// TwinCAT 3 PLC project Fundamentals
// ProgramVersion: 3.1.4023.0
// libraries:
//   Tc2_Standard, * (Beckhoff Automation GmbH)
//   Tc2_System, * (Beckhoff Automation GmbH)
//   Tc2_Utilities, * (Beckhoff Automation GmbH)
//   Tc3_Module, * (Beckhoff Automation GmbH)
// project tree:
//   DUTs/ Breakout.TcDUT
//   DUTs/Simulator/ Compass.TcDUT, Intersection.TcDUT, TrafficDensity.TcDUT, TrafficLight.TcDUT
//   GVLs/ Comparison_GVL.TcGVL, Traffic_GVL.TcGVL
//   / PlcTask.TcTTO
//   POUs/HandsOnProject/ Cars.TcPOU, TrafficManager.TcPOU, TrafficLights.TcPOU
//   POUs/Kim%27s Solution/ Kims_UpdateLights.TcPOU (not stored)
//   POUs/ Ladder.TcPOU, MAIN.TcPOU, StructuredText.TcPOU
// real-time tasks:
//   TASK PlcTask: cycle T#2ms, priority 20, ADS port 350
//   TASK PlcTask1: cycle T#2ms, priority 21, ADS port 351
// I/O:
//   DEVICE Device 1 (EtherCAT), AmsNetId 172.30.193.100.2.1
//     Term 1 (EK1200) [EK1200-5000 EtherCAT Power supply (2A E-Bus)]
//       Term 2 (EL6900) [EL6900, TwinSAFE PLC]
//       Term 3 (EL1904) [EL1904, 4 Ch. Safety Input 24V, TwinSAFE]
//         modules: Module 1 (FSOES)
//       Term 4 (EL2904) [EL2904, 4 Ch. Safety Output 24V, 0.5A, TwinSAFE]
//         modules: Module 1 (FSOES), Module 2 (DO)
//       Term 5 (EL1008) [EL1008 8Ch. Dig. Input 24V, 3ms]
//       Term 6 (EL2008) [EL2008 8Ch. Dig. Output 24V, 0.5A]
//       Term 7 (EL1008) [EL1008 8Ch. Dig. Input 24V, 3ms]
//       Term 8 (EL2008) [EL2008 8Ch. Dig. Output 24V, 0.5A]
//       Term 9 (EL9410) [EL9410 E-Bus Power Supplier  (Diagnostics)]
//       Term 10 (EL1008) [EL1008 8Ch. Dig. Input 24V, 3ms]
//       Term 11 (EL2008) [EL2008 8Ch. Dig. Output 24V, 0.5A]
//       Term 12 (EL1008) [EL1008 8Ch. Dig. Input 24V, 3ms]
//       Term 13 (EL2008) [EL2008 8Ch. Dig. Output 24V, 0.5A]
//       Term 14 (EL1008) [EL1008 8Ch. Dig. Input 24V, 3ms]
//       Term 15 (EL2008) [EL2008 8Ch. Dig. Output 24V, 0.5A]
//       Term 16 (EL9011) [EL9011 End Terminal]
//   DEVICE Device 4 (EtherCAT), AmsNetId 172.30.193.100.5.1
//     Drive 17 (Elmo Drive ) [Gold EtherCAT GCON Drive Rev:0x00010420]
//     Drive 18 (Elmo Drive ) [Gold EtherCAT GCON Drive Rev:0x00010420]
//     Drive 19 (Elmo Drive ) [Gold EtherCAT GCON Drive Rev:0x00010420]
//     Drive 20 (Elmo Drive ) [Gold EtherCAT GCON Drive Rev:0x00010420]
//     Drive 21 (Elmo Drive ) [Gold EtherCAT GCON Drive Rev:0x00010420]
//     Drive 22 (Elmo Drive ) [Gold EtherCAT GCON Drive Rev:0x00010420]

CONFIGURATION Fundamentals
    RESOURCE PLC ON TwinCAT3
        TASK PlcTask(INTERVAL := T#2ms, PRIORITY := 20);
        PROGRAM MAIN WITH PlcTask : MAIN;
    END_RESOURCE
END_CONFIGURATION

// ---- DUTs/Breakout.TcDUT
	{attribute 'OPC.UA.DA' := '1'}
	{attribute 'OPC.UA.DA.StructuredType' := '1'}
TYPE Breakout :
STRUCT
	RedLight	AT %Q*:BOOL; 
	AmberLight	AT %Q*:BOOL;
	GreenLight	AT %Q*:BOOL;
	BlueLight  	AT %Q*:BOOL;
	ButtonPushed AT %I*:BOOL;
END_STRUCT
END_TYPE

// ---- DUTs/Simulator/Compass.TcDUT
{attribute 'strict'}
TYPE Compass :
(
	North:= 1,
	South:= 2,
	East:= 3,
	West:= 4
);
END_TYPE

// ---- DUTs/Simulator/Intersection.TcDUT
	{attribute 'OPC.UA.DA' := '1'}
	{attribute 'OPC.UA.DA.StructuredType' := '1'}
TYPE Intersection :
STRUCT
	NS_Road: TrafficDensity ;//  Values: None/Low/Medium/High
	EW_Road: TrafficDensity ;// Values: None/Low/Medium/High
	
	//The traffic lights facing each direction (N_Light.Red := True -> turns the red light on for traffic flowing North to South);
	N_Light: TrafficLight; //.Red .Amber .Green
	S_Light: TrafficLight; //.Red .Amber .Green
	W_Light: TrafficLight; //.Red .Amber .Green
	E_Light: TrafficLight; //.Red .Amber .Green
	
	//pedestrian crossing request buttons
	N_Ped AT %I*: BOOL;
	S_Ped AT %I*: BOOL;
	E_Ped AT %I*: BOOL;
	W_Ped AT %I*: BOOL;
	
	//Pedestrian safe to cross indicator (the blue light)
	N_Cross AT %Q*: BOOL;
	S_Cross AT %Q*: BOOL;
	E_Cross AT %Q*: BOOL;
	W_Cross AT %Q*: BOOL;
	//Does this direction lead out of the area
	Exit1, Exit2: Compass; //1-4 N S E W
	
	//Stores presense of cars in each direction of the intersection, filled and emptied by the simulation logic
	CarQueue: ARRAY[1..4] OF INT; //1-4 N S E W
END_STRUCT
END_TYPE

// ---- DUTs/Simulator/TrafficDensity.TcDUT
{attribute 'qualified_only'}
{attribute 'OPC.UA.DA' := '1'}
{attribute 'OPC.UA.DA.StructuredType' := '1'}
TYPE TrafficDensity :
(
	None 	:= 0,
	High	:= 1, //Broadway
	Medium	:= 5, //Brick Church
	Low		:= 10 //Fernco
);
END_TYPE

// ---- DUTs/Simulator/TrafficLight.TcDUT
TYPE TrafficLight :
STRUCT
	Red		AT %Q*:BOOL; 
	Amber	AT %Q*:BOOL;
	Green	AT %Q*:BOOL;
END_STRUCT
END_TYPE

// ---- GVLs/Comparison_GVL.TcGVL
{attribute 'qualified_only'} 
VAR_GLOBAL
	NormallyOpen_NO	: BOOL;
	NormallyClosed_NC : BOOL;
	This_And		: BOOL;
	This_Or			: BOOL;
	Or_This			: BOOL;
	Or_NOT_This		: BOOL:=TRUE;
	But_NOT_This	: BOOL:=TRUE;
	And_This		: BOOL;
	Tada			: BOOL;
	OffTimer_TOF	: TOF;
	OnTimer_TON		: TON;
	PulseTimer_TP	: TP;
	TurnOFFAfter	: BOOL;
	TurnONAfter		: BOOL;
	TurnOnFor		: BOOL;
	DefaultON		: BOOL;
	DefaultOFF		: BOOL;
	Countdown		: CTD;
	
	CountUP			: CTU;
	CountTo25		: BOOL;
END_VAR
VAR_GLOBAL CONSTANT
	DURATION		:TIME:=T#15S;
	SHORT_DURATION	:TIME:=T#5S;
END_VAR

// ---- GVLs/Traffic_GVL.TcGVL
VAR_GLOBAL
	{attribute 'OPC.UA.DA' := '1'}
	{attribute 'OPC.UA.DA.StructuredType' := '1'}
	FirstAndMain 	:Intersection;
	{attribute 'OPC.UA.DA' := '1'}
	{attribute 'OPC.UA.DA.StructuredType' := '1'}
	SecondAndMain 	:Intersection;
	{attribute 'OPC.UA.DA' := '1'}
	{attribute 'OPC.UA.DA.StructuredType' := '1'}
	FirstAndPine	:Intersection;
	{attribute 'OPC.UA.DA' := '1'}
	{attribute 'OPC.UA.DA.StructuredType' := '1'}
	SecondAndPine	:Intersection;
	
END_VAR

// ---- POUs/MAIN.TcPOU
PROGRAM MAIN
VAR
	ClimbTheRungs, MoveOnToCode, PlayInTraffic, RunOnce:BOOL:=FALSE;
	
	{attribute 'OPC.UA.DA' := '1'}
	{attribute 'OPC.UA.DA.StructuredType' := '1'}
	FirstSteps:Breakout;
END_VAR

// <- this is how you comment out lines, anything after the // will not be part of the program 
//this is how you can leave notes for future developers or if code isn't working right you can remove it temporarily to test things without deleting it  

//THIS SPACE IS WHERE YOU CAN PUT YOUR FIRST CODE, Try removing the // from the next line
//FirstSteps.BlueLight := TRUE;


IF ClimbTheRungs THEN
	Ladder(); //This calls the ladder logic example
ELSIF MoveOnToCode THEN
StructuredText(); //This calls the structured text example
ELSIF PlayInTraffic THEN
	IF NOT RunOnce THEN
	TrafficManager.Init();
	runOnce:=TRUE;
END_IF
TrafficManager.Update();
END_IF

END_PROGRAM

// ---- POUs/Ladder.TcPOU
PROGRAM Ladder
VAR

END_VAR
VAR // added by the converter: edge detectors and wires of the graphical bodies
    _rt1 : R_TRIG;
END_VAR

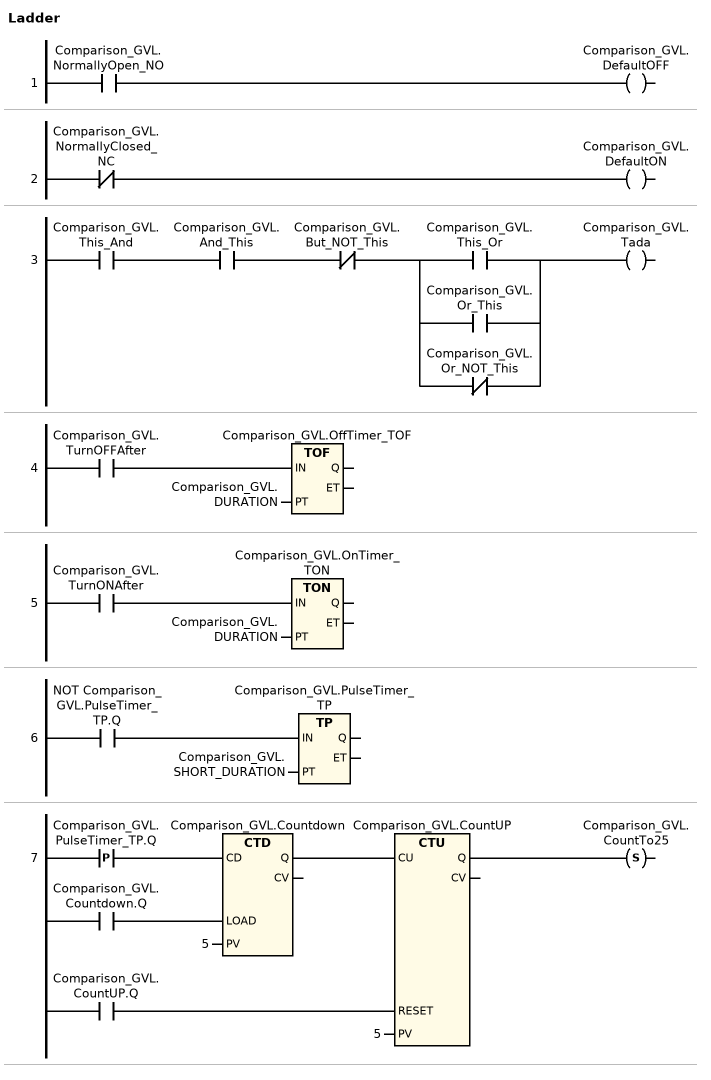
// NETWORK 1
Comparison_GVL.DefaultOFF := Comparison_GVL.NormallyOpen_NO;

// NETWORK 2
Comparison_GVL.DefaultON := NOT Comparison_GVL.NormallyClosed_NC;

// NETWORK 3
Comparison_GVL.Tada := Comparison_GVL.This_And AND Comparison_GVL.And_This AND NOT Comparison_GVL.But_NOT_This AND (Comparison_GVL.This_Or OR Comparison_GVL.Or_This OR NOT Comparison_GVL.Or_NOT_This);

// NETWORK 4
Comparison_GVL.OffTimer_TOF(IN := Comparison_GVL.TurnOFFAfter, PT := Comparison_GVL.DURATION); // TOF

// NETWORK 5
Comparison_GVL.OnTimer_TON(IN := Comparison_GVL.TurnONAfter, PT := Comparison_GVL.DURATION); // TON

// NETWORK 6
Comparison_GVL.PulseTimer_TP(IN := NOT Comparison_GVL.PulseTimer_TP.Q, PT := Comparison_GVL.SHORT_DURATION); // TP

// NETWORK 7
_rt1(CLK := Comparison_GVL.PulseTimer_TP.Q);
Comparison_GVL.Countdown(CD := _rt1.Q, LOAD := Comparison_GVL.Countdown.Q, PV := 5); // CTD
Comparison_GVL.CountUP(CU := Comparison_GVL.Countdown.Q, RESET := Comparison_GVL.CountUP.Q, PV := 5); // CTU
Comparison_GVL.CountTo25 S= Comparison_GVL.CountUP.Q;

END_PROGRAM

// ---- POUs/StructuredText.TcPOU
PROGRAM StructuredText
VAR
	ChangeTime		:TIME:=T#1S;
	CountOnes		:INT:=1;
	CountFives		:INT:=1;
	JustOncePer 	:R_TRIG;
	DidSomething:BOOL;
	AlsoCountTo25	: BOOL;
END_VAR
VAR CONSTANT
	ST_DURATION	:TIME:=T#2S;
END_VAR

	Comparison_GVL.DefaultOFF	:=	Comparison_GVL.NormallyOpen_NO; //Sets DefaultOFF equal to whatever NormallyOpen is set to
	Comparison_GVL.DefaultON	:=	NOT Comparison_GVL.NormallyClosed_NC; //Sets DefaultON equal to the opposite of what NormallyClosed is set to
	
	Comparison_GVL.Tada			:= Comparison_GVL.This_And AND Comparison_GVL.And_This	AND NOT Comparison_GVL.But_NOT_This	AND
								(Comparison_GVL.This_Or OR Comparison_GVL.Or_This OR NOT Comparison_GVL.Or_NOT_This);
	
	// this line ^ and this next one technically do the same thing BUT if I wanted to do more complicated stuff or multiple things I need to use the IF 
	
	IF Comparison_GVL.This_And AND Comparison_GVL.And_This	AND NOT Comparison_GVL.But_NOT_This	AND
		(Comparison_GVL.This_Or OR Comparison_GVL.Or_This OR NOT Comparison_GVL.Or_NOT_This) THEN
		Comparison_GVL.Tada	:= TRUE;
	ELSE
		Comparison_GVL.Tada	:= FALSE;
	END_IF
	
	Comparison_GVL.OffTimer_TOF(IN:=Comparison_GVL.TurnOFFAfter,PT:= ST_DURATION);
	Comparison_GVL.OnTimer_TON(IN:=Comparison_GVL.TurnONAfter,PT:= ST_DURATION);
	Comparison_GVL.PulseTimer_TP(IN:=NOT Comparison_GVL.PulseTimer_TP.Q,PT:= ChangeTime);
	JustOncePer(CLK:= Comparison_GVL.PulseTimer_TP.Q);
	
	IF JustOncePer.Q THEN
		CountOnes:= CountOnes+1;
		Comparison_GVL.TurnOnFor:=FALSE;
	END_IF
	IF CountOnes = 5 THEN
		CountFives:= CountFives +1;
		CountOnes:=1;
	END_IF	
	
	DidSomething:= DoSomething(Counter:= (CountOnes*CountFives) );
	
	IF CountFives = 5 THEN
		CountFives:=1;
	END_IF

METHOD DoSomething : BOOL
VAR_INPUT
	Counter:INT;
END_VAR
CASE Counter OF
	1,10,20:
		Comparison_GVL.TurnOFFAfter:=TRUE;
		Comparison_GVL.TurnONAfter:=TRUE;
		DoSomething:=TRUE;
	2,11,21:
		Comparison_GVL.TurnOFFAfter:=FALSE;
		DoSomething:=TRUE;
	3:
		Comparison_GVL.This_And:=TRUE;
		Comparison_GVL.And_This:=TRUE;
		DoSomething:=TRUE;
	5:
		Comparison_GVL.But_NOT_This:=FALSE;
		DoSomething:=TRUE;
	7:
		Comparison_GVL.This_Or:=TRUE;
		DoSomething:=TRUE;
	9,19:
		Comparison_GVL.TurnONAfter:=FALSE;
		DoSomething:=TRUE;
	13:
		Comparison_GVL.Or_This:=TRUE;
		DoSomething:=TRUE;
	15:
		Comparison_GVL.Or_This:=FALSE;
		Comparison_GVL.Or_NOT_This:=FALSE;
		DoSomething:=TRUE;
	17:
		Comparison_GVL.This_Or:=FALSE;
		Comparison_GVL.Or_This:=FALSE;
		DoSomething:=TRUE;
	25:
		AlsoCountTo25:=TRUE;
	ELSE
		DoSomething:=FALSE;
		Comparison_GVL.TurnOnFor:=TRUE;
END_CASE
END_METHOD

END_PROGRAM

// ---- POUs/HandsOnProject/TrafficManager.TcPOU
PROGRAM TrafficManager
VAR
Simulator: Cars;
UpdateLights: Kims_UpdateLights;
runOnce:BOOL:=FALSE;
END_VAR

METHOD Change_TrafficFlow : BOOL
VAR_INPUT
	Intersect: POINTER to Intersection;
	NewNS_Density, NewEW_Density: TrafficDensity;
	Exit1, Exit2: Compass;
END_VAR
Intersect^.NS_Road:= NewNS_Density;
Intersect^.EW_Road:= NewEW_Density;
Intersect^.Exit1 := Exit1;
Intersect^.Exit2 := Exit2;
END_METHOD

METHOD Init : BOOL
VAR_INPUT
	//First, Second, Main, Pine :TrafficDensity;
END_VAR
//FirstAndMain.NS_Road:=TrafficDensity.Low;
//FirstAndMain.EW_Road:=TrafficDensity.Medium;
//FirstAndMain.Exit1:= North;
//FirstAndMain.Exit2:= West;
Change_TrafficFlow(ADR(FirstAndMain),TrafficDensity.Low,TrafficDensity.Medium, North, West);
Change_TrafficFlow(ADR(SecondAndMain),TrafficDensity.Medium,TrafficDensity.Medium, North, East);

Change_TrafficFlow(ADR(FirstAndPine),TrafficDensity.Low,TrafficDensity.High, South, West);
Change_TrafficFlow(ADR(SecondAndPine),TrafficDensity.Medium,TrafficDensity.High, South, East);
END_METHOD

METHOD Update
VAR_INPUT
END_VAR
UpdateLights(Intersect:=ADR(FirstAndMain));
UpdateLights(Intersect:=ADR(SecondAndMain));
//			  |						   |
//---------------<-Main Street->------------------
//		First |					Second |
//			  |						   |
//			  |  					   |
//----------------<-Pine Street->------------------
//			  |						   |
UpdateLights(Intersect:=ADR(FirstAndPine));
UpdateLights(Intersect:=ADR(SecondAndPine));


//Below this point I'm just Playing with my Hot Wheels haha//
Simulator.AddCars(ADR(FirstAndMain));
Simulator.AddCars(ADR(SecondAndMain));
Simulator.AddCars(ADR(FirstAndPine));
Simulator.AddCars(ADR(SecondAndPine));
Simulator.MoveCars(ADR(FirstAndMain), ADR(SecondAndMain), Compass.East, ADR(FirstAndPine), Compass.South);
Simulator.MoveCars(ADR(SecondAndPine), ADR(SecondAndMain), Compass.North, ADR(FirstAndPine), Compass.West);
END_METHOD

END_PROGRAM

// ---- POUs/HandsOnProject/Cars.TcPOU
FUNCTION_BLOCK Cars
VAR_INPUT
END_VAR
VAR_OUTPUT
END_VAR
VAR
	CarSpawner		:TON;
	SpawnRate		:INT;
END_VAR

METHOD AddCars : BOOL
VAR_INPUT
	Intersect:POINTER TO Intersection;
END_VAR
VAR
	Frequency: TIME := T#1S;
END_VAR
CarSpawner(IN := NOT CarSpawner.Q, PT := Frequency);
IF CarSpawner.Q THEN
	SpawnRate:=SpawnRate+1;
	CASE Intersect^.Exit1 OF
		North, South:
			IF SpawnRate MOD Intersect^.NS_Road = 0 THEN
				Intersect^.CarQueue[Intersect^.Exit1]:= Intersect^.CarQueue[Intersect^.Exit1] +1;
			END_IF		
		East, West:
			IF SpawnRate MOD Intersect^.EW_Road = 0 THEN
				Intersect^.CarQueue[Intersect^.Exit1]:= Intersect^.CarQueue[Intersect^.Exit1] +1;
			END_IF
	END_CASE
	IF NOT (Intersect^.Exit2 = Intersect^.Exit1) THEN
		CASE Intersect^.Exit2 OF	
		North, South:
			IF SpawnRate MOD Intersect^.NS_Road = 0 THEN
				Intersect^.CarQueue[Intersect^.Exit2]:= Intersect^.CarQueue[Intersect^.Exit2] +1;
			END_IF		
		East, West:
			IF SpawnRate MOD Intersect^.EW_Road = 0 THEN
				Intersect^.CarQueue[Intersect^.Exit2]:= Intersect^.CarQueue[Intersect^.Exit2] +1;
			END_IF
		END_CASE	
	END_IF

END_IF
IF SpawnRate = 10 THEN
	SpawnRate :=0;
END_IF
END_METHOD

METHOD MoveCars : BOOL
VAR_INPUT
	To_Intersect, From_A: POINTER TO Intersection;
	Direction_A: Compass;
	From_B: POINTER TO Intersection;
 	Direction_B: Compass;	
END_VAR
//The traffic lights are facing each direction (N_Light.Red := True -> turns the red light facing north on stopping traffic flowing North to South);
IF CarSpawner.Q THEN
	CASE Direction_A OF
	North:
		IF From_A^.N_Light.Green = TRUE AND From_A^.CarQueue[North]>0 THEN
			From_A^.CarQueue[North]:= From_A^.CarQueue[North] - 1;
			IF To_Intersect^.N_Light.Green AND (To_Intersect^.Exit1 = North OR To_Intersect^.Exit2 = North) THEN
				To_Intersect^.CarQueue[North]:= To_Intersect^.CarQueue[North] - 1;
			ELSE
				To_Intersect^.CarQueue[North]:= To_Intersect^.CarQueue[North] + 1;
			END_IF
			
		END_IF
		IF To_Intersect^.S_Light.Green = TRUE AND To_Intersect^.CarQueue[South]>0 THEN
			To_Intersect^.CarQueue[South]:= To_Intersect^.CarQueue[South] - 1;
			IF From_A^.S_Light.Green AND (From_A^.Exit1 = South OR From_A^.Exit2 = South) THEN
				From_A^.CarQueue[South]:= From_A^.CarQueue[South] - 1;
			ELSE
				From_A^.CarQueue[South]:= From_A^.CarQueue[South] + 1;
			END_IF
		END_IF
	South:
		IF From_A^.S_Light.Green = TRUE AND From_A^.CarQueue[South]>0 THEN
			From_A^.CarQueue[South]:= From_A^.CarQueue[South] - 1;
			IF To_Intersect^.S_Light.Green AND (To_Intersect^.Exit1 = South OR To_Intersect^.Exit2 = South) THEN
				To_Intersect^.CarQueue[South]:= To_Intersect^.CarQueue[South] - 1;
			ELSE
				To_Intersect^.CarQueue[South]:= To_Intersect^.CarQueue[SOuth] + 1;
			END_IF
			
		END_IF
		IF To_Intersect^.N_Light.Green = TRUE AND To_Intersect^.CarQueue[North]>0 THEN
			To_Intersect^.CarQueue[North]:= To_Intersect^.CarQueue[North] - 1;
			IF From_A^.N_Light.Green AND (From_A^.Exit1 = North OR From_A^.Exit2 = North) THEN
				From_A^.CarQueue[North]:= From_A^.CarQueue[North] - 1;
			ELSE
				From_A^.CarQueue[North]:= From_A^.CarQueue[North] + 1;
			END_IF
		END_IF
	East:
		IF From_A^.E_Light.Green = TRUE AND From_A^.CarQueue[East]>0 THEN
			From_A^.CarQueue[East]:= From_A^.CarQueue[East] - 1;
			IF To_Intersect^.E_Light.Green AND (To_Intersect^.Exit1 = East OR To_Intersect^.Exit2 = East) THEN
				To_Intersect^.CarQueue[East]:= To_Intersect^.CarQueue[East] - 1;
			ELSE
				To_Intersect^.CarQueue[East]:= To_Intersect^.CarQueue[East] + 1;
			END_IF
			
		END_IF
		IF To_Intersect^.W_Light.Green = TRUE AND To_Intersect^.CarQueue[West]>0 THEN
			To_Intersect^.CarQueue[West]:= To_Intersect^.CarQueue[West] - 1;
			IF From_A^.W_Light.Green AND (From_A^.Exit1 = West OR From_A^.Exit2 = West) THEN
				From_A^.CarQueue[West]:= From_A^.CarQueue[West] - 1;
			ELSE
				From_A^.CarQueue[West]:= From_A^.CarQueue[West] + 1;
			END_IF
		END_IF
	West:
		IF From_A^.W_Light.Green = TRUE AND From_A^.CarQueue[West]>0 THEN
			From_A^.CarQueue[West]:= From_A^.CarQueue[West] - 1;
			IF To_Intersect^.W_Light.Green AND (To_Intersect^.Exit1 = West OR To_Intersect^.Exit2 = West) THEN
				To_Intersect^.CarQueue[West]:= To_Intersect^.CarQueue[West] - 1;
			ELSE
				To_Intersect^.CarQueue[West]:= To_Intersect^.CarQueue[West] + 1;
			END_IF
			
		END_IF
		IF To_Intersect^.E_Light.Green = TRUE AND To_Intersect^.CarQueue[East]>0 THEN
			To_Intersect^.CarQueue[East]:= To_Intersect^.CarQueue[East] - 1;
			IF From_A^.E_Light.Green AND (From_A^.Exit1 = East OR From_A^.Exit2 = East) THEN
				From_A^.CarQueue[East]:= From_A^.CarQueue[East] - 1;
			ELSE
				From_A^.CarQueue[East]:= From_A^.CarQueue[East] + 1;
			END_IF
		END_IF
	END_CASE
		CASE Direction_B OF
	North:
		IF From_B^.N_Light.Green = TRUE AND From_B^.CarQueue[North]>0 THEN
			From_B^.CarQueue[North]:= From_B^.CarQueue[North] - 1;
			IF To_Intersect^.N_Light.Green AND (To_Intersect^.Exit1 = North OR To_Intersect^.Exit2 = North) THEN
				To_Intersect^.CarQueue[North]:= To_Intersect^.CarQueue[North] - 1;
			ELSE
				To_Intersect^.CarQueue[North]:= To_Intersect^.CarQueue[North] + 1;
			END_IF
			
		END_IF
		IF To_Intersect^.S_Light.Green = TRUE AND To_Intersect^.CarQueue[South]>0 THEN
			To_Intersect^.CarQueue[South]:= To_Intersect^.CarQueue[South] - 1;
			IF From_B^.S_Light.Green AND (From_B^.Exit1 = South OR From_B^.Exit2 = South) THEN
				From_B^.CarQueue[South]:= From_B^.CarQueue[South] - 1;
			ELSE
				From_B^.CarQueue[South]:= From_B^.CarQueue[South] + 1;
			END_IF
		END_IF
	South:
		IF From_B^.S_Light.Green = TRUE AND From_B^.CarQueue[South]>0 THEN
			From_B^.CarQueue[South]:= From_B^.CarQueue[South] - 1;
			IF To_Intersect^.S_Light.Green AND (To_Intersect^.Exit1 = South OR To_Intersect^.Exit2 = South) THEN
				To_Intersect^.CarQueue[South]:= To_Intersect^.CarQueue[South] - 1;
			ELSE
				To_Intersect^.CarQueue[South]:= To_Intersect^.CarQueue[SOuth] + 1;
			END_IF
			
		END_IF
		IF To_Intersect^.N_Light.Green = TRUE AND To_Intersect^.CarQueue[North]>0 THEN
			To_Intersect^.CarQueue[North]:= To_Intersect^.CarQueue[North] - 1;
			IF From_B^.N_Light.Green AND (From_B^.Exit1 = North OR From_B^.Exit2 = North) THEN
				From_B^.CarQueue[North]:= From_B^.CarQueue[North] - 1;
			ELSE
				From_B^.CarQueue[North]:= From_B^.CarQueue[North] + 1;
			END_IF
		END_IF
	East:
		IF From_B^.E_Light.Green = TRUE AND From_B^.CarQueue[East]>0 THEN
			From_B^.CarQueue[East]:= From_B^.CarQueue[East] - 1;
			IF To_Intersect^.E_Light.Green AND (To_Intersect^.Exit1 = East OR To_Intersect^.Exit2 = East) THEN
				To_Intersect^.CarQueue[East]:= To_Intersect^.CarQueue[East] - 1;
			ELSE
				To_Intersect^.CarQueue[East]:= To_Intersect^.CarQueue[East] + 1;
			END_IF
			
		END_IF
		IF To_Intersect^.W_Light.Green = TRUE AND To_Intersect^.CarQueue[West]>0 THEN
			To_Intersect^.CarQueue[West]:= To_Intersect^.CarQueue[West] - 1;
			IF From_B^.W_Light.Green AND (From_B^.Exit1 = West OR From_B^.Exit2 = West) THEN
				From_B^.CarQueue[West]:= From_B^.CarQueue[West] - 1;
			ELSE
				From_B^.CarQueue[West]:= From_B^.CarQueue[West] + 1;
			END_IF
		END_IF
	West:
		IF From_B^.W_Light.Green = TRUE AND From_B^.CarQueue[West]>0 THEN
			From_B^.CarQueue[West]:= From_B^.CarQueue[West] - 1;
			IF To_Intersect^.W_Light.Green AND (To_Intersect^.Exit1 = West OR To_Intersect^.Exit2 = West) THEN
				To_Intersect^.CarQueue[West]:= To_Intersect^.CarQueue[West] - 1;
			ELSE
				To_Intersect^.CarQueue[West]:= To_Intersect^.CarQueue[West] + 1;
			END_IF
			
		END_IF
		IF To_Intersect^.E_Light.Green = TRUE AND To_Intersect^.CarQueue[East]>0 THEN
			To_Intersect^.CarQueue[East]:= To_Intersect^.CarQueue[East] - 1;
			IF From_B^.E_Light.Green AND (From_B^.Exit1 = East OR From_B^.Exit2 = East) THEN
				From_B^.CarQueue[East]:= From_B^.CarQueue[East] - 1;
			ELSE
				From_B^.CarQueue[East]:= From_B^.CarQueue[East] + 1;
			END_IF
		END_IF
	END_CASE
	
END_IF
END_METHOD

END_FUNCTION_BLOCK

// ---- POUs/HandsOnProject/TrafficLights.TcPOU
FUNCTION_BLOCK TrafficLights
VAR_INPUT
END_VAR
VAR_OUTPUT
END_VAR
VAR
END_VAR

//This is where all the stuff you guys are going to add will go.

END_FUNCTION_BLOCK
